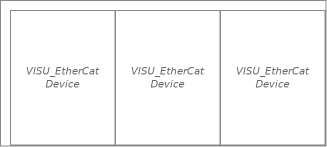
VISUALIZATION VISU_ServicesTimingIO  // 327x147
VAR_IN_OUT
	ref : ServicesTimingIO;
    widget : ServicesTimingIOWidget;
END_VAR
    Frame (10,10 105x135)
        shows VISU_EtherCatDevice(device := ref.parts.coupler, widget := widget.coupler)
    Frame (115,10 105x135)
        shows VISU_EtherCatDevice(device := ref.parts.slot1, widget := widget.slot1)
    Frame (220,10 105x135)
        shows VISU_EtherCatDevice(device := ref.parts.slot2, widget := widget.slot2)
END_VISUALIZATION

(* stored: Version 1.1.0.1, ProductVersion 3.1.4019.2
   Visu VISU_ServicesTimingIO: Id {65bf82ce-aed9-4182-9e0b-9c6a2c2af0ab} *)
